// TwinCAT 3 PLC project EL6851_DMX
// ProgramVersion: 3.1.4023.0
// libraries:
//   Tc2_DMX, * (Beckhoff Automation GmbH)
//   Tc2_Standard, * (Beckhoff Automation GmbH)
//   Tc2_System, * (Beckhoff Automation GmbH)
//   Tc3_Module, * (Beckhoff Automation GmbH)
// project tree:
//   / PlcTask.TcTTO
//   POUs/ MAIN.TcPOU, P_DMX_Master.TcPOU, P_DMX_Slave.TcPOU

CONFIGURATION EL6851_DMX
    RESOURCE PLC ON TwinCAT3
        TASK PlcTask(INTERVAL := T#10ms, PRIORITY := 24);
        PROGRAM MAIN WITH PlcTask : MAIN;
    END_RESOURCE
END_CONFIGURATION

// ---- POUs/MAIN.TcPOU
PROGRAM MAIN
VAR
END_VAR

P_DMX_Master();
P_DMX_Slave();

END_PROGRAM

// ---- POUs/P_DMX_Master.TcPOU
PROGRAM P_DMX_Master
VAR
	(*	As a default only the output channels 1-512 are activated in the process image of the DMX Master terminal (EL6851)
		this can be modified in the tab "Process Data" of the terminal:
			* if less channels are wanted,
			* if RDM communication is wanted, the input channels also have to be enabled and linked.
	*)
	DMX_Master_In		AT %I*	: ST_EL6851InDataEx;	
	DMX_Master_Out		AT %Q*	: ST_EL6851OutData;	

	fbCommunication				: FB_EL6851CommunicationEx;
	stCommandBuffer				: ST_DMXCommandBuffer;
	arrProcessData				: ARRAY [1..512] OF BYTE;
END_VAR

// Communication
// =============
fbCommunication(
	wSourceManufacturerId		:= 16#42_41, 
	dwSourceDeviceId			:= 16#12_13_14_15, 
	bEnableSendingData			:= TRUE, 
	bSetCycleMode				:= TRUE, 
	bSendDefaultData			:= FALSE, 
	uiDataLength				:= 512, 
	dwOptions					:= , 
	bError						=> , 
	udiErrorId					=> , 
	bCycleMode					=> , 
	byBufferDemandMeter			=> , 
	byBufferMaximumDemandMeter	=> , 
	uiBufferOverflowCounter		=> , 
	bLineIsBusy					=> , 
	stEL6851InData				:= DMX_Master_In, 
	stEL6851OutData				:= DMX_Master_Out, 
	stCommandBuffer				:= stCommandBuffer, 
	arrProcessData				:= arrProcessData);
	
// Controlling DMX addresses (without RDM)
// =======================================
// To send values to the DMX network, it is sufficient to write the wanted value in the " arrProcessData" using the address as the array index. 

arrProcessData[12]	:= 221;	// Sends the value 221 to DMX address 12

arrProcessData[57]	:= 0;	// Sends the value 0 to DMX address 57

// for examples on controlling DMX devices via RDM
// ===============================================
// Please use the example described in the link below or contact Beckhoff
// https://infosys.beckhoff.com/content/1033/tcplclibdmx/html/sample02.htm?id=1245473112320324804

END_PROGRAM

// ---- POUs/P_DMX_Slave.TcPOU
PROGRAM P_DMX_Slave
VAR
	(*	As a default only channels 1-64 are activated in the process image of the DMX Slave terminal (EL6851-0010)
		If more or other channels are wanted, this can be modified in the tab "Process Data" of the terminal:
	*)

	DMX_Slave_In		AT %I*	: ARRAY[1..64] OF BYTE;
		
END_VAR

(*	The data received from the DMX network can be found in the array linked to the peripheral data range from the terminal in the corresponding index 
	and the value can be used in the PLC program as needed.

*)

DMX_Slave_In[7];	(* Contains the data for Channel 7 in the received DMX telegram *) 

DMX_Slave_In[35];	(* Contains the data for Channel 35 in the received DMX telegram *)

END_PROGRAM
